{attribute 'GeneratedUsingTerminal: AT2041-0250-0022'}
{attribute addProperty BoxType "AT2041-0250-0022"}
{attribute addProperty Id "A_0100_AT2040_5250_0019_AT2040_5250AT2040_33A3DF1B80"}
{attribute addProperty CRC "1520056762"}
{attribute addProperty Size "80"}
TYPE A_0044_AT2041_0250_0022_5A9A39BA EXTENDS AT2041_2EA6C9BF :
STRUCT
	{attribute addProperty Name "A_0100_AT2040_5250_0019_AT2040_5250"}
	A_0100_AT2040_5250_0019_AT2040_5250 : AT2040_33A3DF1B;
END_STRUCT
END_TYPE

(* stored: Version 1.2.0.0, ProductVersion 3.1.4024.9
   DUT A_0044_AT2041_0250_0022_5A9A39BA: Id {01b4b0f1-9577-4e01-a7c4-ae86b1f29e43} *)
